# B&R Automation Studio project Masdgrt
Automation Studio 4.9

## Configuration ConfigSortingSystem

### Task classes (Cpu.sw)
```
Cyclic#4:
  Program <- Program.prg
  Program3R4 <- Program3R4TG.prg
Libraries: McBase, MpAxis, McAxis, MpBase, McAcpAx, CoTrace, AsZip, FileIO, runtime
```

## Logical view

### Global.var - Global variables
```iecst
VAR
	ZmiennaGlobalnaBartasa : INT;
	ZmiennaGlobalnaBartasa2 : USINT;
END_VAR
```

- Visualisation Logical/mappView (not shown)

### Program Logical/Program (IEC)

#### Variables.var
```iecst
VAR
	MotorBeltAxisBasic : MpAxisBasic;
	MotorBeltParType : MpAxisBasicParType;
	BAIT : UINT;
	Wysun : BOOL;
	Moja_zmienna_szymon : BOOL;
END_VAR
```

#### Main.st
```iecst
PROGRAM _INIT
	//BARTAS
	//BARTAS
	//Wysun; // testowa zmienna

END_PROGRAM

PROGRAM _CYCLIC
	//przesuwam program SZYMON
	//BARTAS
//	IF Wysun THEN  //TESTOWANIE
//		BAIT := 2#0000_0000_0000_0101;
//	ELSE
//		BAIT := 2#0000_0000_0000_0000;
//	END_IF;
	IF Zmienna THEN
		Zmienna := 0;
	END_IF;
	IF Zmienna THEN
		Zmienna := 0;
		IF Zmienna THEN
			Zmienna := 0;
		END_IF;
	END_IF;
	//Fragment kodu odpowiedzialny za inicjalizacjê taœmy
	gAxis_1;
	MotorBeltAxisBasic.MpLink := ADR(gAxis_1);
	MotorBeltAxisBasic.Enable := TRUE;
	MotorBeltAxisBasic.Parameters := ADR(MotorBeltParType);
	MotorBeltAxisBasic();
	IF Zmienna THEN
		Zmienna := 0;
	END_IF;
	//Zmieniam coœ

	IF BAIT THEN
		ZmiennaGlobalnaBartasa2 := 1;
	END_IF;

	IF Wysun THEN
		ZmiennaGlobalnaBartasa := 10;
		IF ZmiennaGlobalnaBartasa = 10 THEN
	  		BAIT := 2#0000_0000_0000_0000;
		END_IF;
	END_IF;

	//LOL

	//dupa
END_PROGRAM

PROGRAM _EXIT
	//BARTAS 2

	//BARTAS 2
	 	//BARTAS
END_PROGRAM
```

Listed in the project but not available here: Logical/Global.typ, Logical/Libraries, Logical/ZRODLODRZEWO
